FUNCTION_BLOCK FB_Machine EXTENDS FB_Generic
VAR_INPUT
	pPML_Instance1	: POINTER TO FB_Generic;
	pPML_Instance2	: POINTER TO FB_Generic;//instance for couple and uncouple
	pPackTags		: POINTER TO ST_PackMLv30;
	pSafetySystem	: POINTER TO FB_Safety_Subsystem;
END_VAR
VAR_OUTPUT

END_VAR
VAR	
	stSubModuleInfo		: ARRAY [1..iSubModule] OF ST_PMLSubUnitInfo;	//Informations about the Subunits
//	pPML_Instance	: ARRAY [1..iSubModule] OF POINTER TO FB_Generic;
	arrCouple	: ARRAY [1..iSubModule] OF BOOL;
	arrCmd		: ARRAY [1..iSubModule] OF E_PMLCommand;
	unCouple	: BOOL;//all modules uncoupling
	
	rtrig_alarm	:ARRAY [1..iSubModule] OF ARRAY[1..MaxAlarms] OF R_TRIG;
	
	iCmd_unitsActive	: INT;
	iCmd_transfer	: INT;


	preEstate	: E_PMLState;
	
END_VAR
VAR CONSTANT
	iSubModule	: UINT :=2;
END_VAR

//pPML_Instance[1]	:= ADR(GVL.fb_sample1);
//pPML_Instance[2]	:= ADR(GVL.fb_sample2);
///////////////////////////////////////////for signal system/////////////////////////////////////////////////////////////
IF NOT unCouple THEN
	FOR i:=1 TO UINT_TO_INT(iSubModule) DO
		arrCmd[i]:=eCommand;
		arrCouple[i]:= TRUE;
//		pPML_Instance[i]^._bCouple	:= TRUE;

	END_FOR
END_IF
unCouple	:= TRUE;//for mix sysytem
//////////////////////////////////////////////couple cmd//////////////////////////////////////////////////////////
//FOR i:=1 TO UINT_TO_INT(iSubModule) DO
//	IF arrCouple[i] THEN
//		arrCmd[i]:=eCommand;
//	END_IF
//END_FOR

CASE iCmd_transfer OF	
	0:
		IF eCommand<>ePMLCommand_Undefined THEN
			iCmd_transfer	:= 1;
		END_IF
	1:	
		IF arrCouple[1] THEN
			arrCmd[1]	:= eCommand;
		END_IF
		IF arrCouple[2] THEN
			arrCmd[2]	:= eCommand;
		END_IF
		iCmd_transfer	:= 2;	
	2:
		CASE preEstate OF
			ePMLState_Undefined:
				IF eState=ePMLState_Aborted THEN
					iCmd_transfer	:= 3;
				END_IF			
			ePMLState_Aborted,ePMLState_Clearing:
				IF eState=ePMLState_Stopped OR eState=ePMLState_Aborted THEN
					iCmd_transfer	:= 3;
				END_IF
			ePMLState_Stopped,ePMLState_Resetting:
				IF eState=ePMLState_Idle OR eState=ePMLState_Aborted THEN
					iCmd_transfer	:= 3;
				END_IF				
			ePMLState_Idle,ePMLState_Starting:
				IF eState=ePMLState_Execute OR eState=ePMLState_Stopped OR eState=ePMLState_Aborted THEN
					iCmd_transfer	:= 3;
				END_IF				
			ePMLState_Execute,ePMLState_Aborting,ePMLState_Stopping:
				IF eState=ePMLState_Stopped OR eState=ePMLState_Aborted THEN
					iCmd_transfer	:= 3;
				END_IF				
		END_CASE	
	3:
		arrCouple[2]	:= FALSE;
		arrCmd[1]	:=	ePMLCommand_Undefined;
		arrCmd[2]	:=	ePMLCommand_Undefined;
		iCmd_transfer	:= 0;	
END_CASE



pPML_Instance1^(
	eModeCommand:= eModeCommand, 
	eCommand:= arrCmd[1], 
	eMode=> , 
	eState=> stSubModuleInfo[1].eState, 
	bUndefinedDone=> , 
	bInvalidModeCommandOut=> , 
	bChangeIntoProduction=> );
stSubModuleInfo[1].Active		:= arrCouple[1];

pPML_Instance2^(
	eModeCommand:= eModeCommand, 
	eCommand:= , 
	eMode=> , 
	eState=> stSubModuleInfo[2].eState, 
	bUndefinedDone=> , 
	bInvalidModeCommandOut=> , 
	bChangeIntoProduction=> );
IF stSubModuleInfo[2].Active THEN
	pPML_Instance2^.eCommand	:= arrCmd[2];
END_IF	
stSubModuleInfo[2].Active		:= arrCouple[2];


IF  pPML_Instance1^.bUndefinedDone AND 
	pPML_Instance2^.bUndefinedDone 
THEN
	bUndefinedDone := TRUE;
END_IF

//The fbStateMachine from FB_Machine gets the Information about the states and activity from the subunits
fbStateMachine.stSubUnitInfoRef.ArraySize		:= SIZEOF(stSubModuleInfo);
fbStateMachine.stSubUnitInfoRef.NoOfSubUnits	:= iSubModule;
fbStateMachine.stSubUnitInfoRef.pArray			:= ADR(stSubModuleInfo);



//Set unit information 
M_SetUnitInfo();






SUPER^();

{attribute 'object_name' := 'M_Clearing'}
METHOD M_Clearing

CASE fbUnitModeManager.eModeStatus OF
	ePMLProtUnitMode_Production:		//Production, Mantainance, Manual
		FOR i:=1 TO 3 DO//try clear alarm several times
			FOR j:=1 TO MaxAlarms DO
				GVL.pml_adminAlarm.M_AcknowledgeAlarm(stAdmin:=pPackTags^.Admin,stAlarm:=pPackTags^.Admin.Alarm[j]);
				GVL.pml_adminAlarm.M_ClearAlarm(stAdmin:=pPackTags^.Admin,stAlarm:=pPackTags^.Admin.Alarm[j]);
			END_FOR	
		END_FOR	
		IF pSafetySystem^.M_reset() THEN
			IF pSafetySystem^.xError THEN
				IF M_UnitsActive(ePMLCommand_Abort)THEN
					eCommand	:= ePMLCommand_Abort;
				END_IF
			ELSE
				M_StateComplete();
			END_IF
		END_IF	
		
	
	ePMLProtUnitMode_Maintenance, ePMLProtUnitMode_Manual, ePMLUnitMode_Service:
		M_StateComplete();
END_CASE
END_METHOD

{attribute 'object_name' := 'M_Execute'}
METHOD M_Execute
END_METHOD

{attribute 'object_name' := 'M_Resetting'}
METHOD M_Resetting
CASE fbUnitModeManager.eModeStatus OF
	ePMLProtUnitMode_Production:		//Production, Mantainance, Manual	
		IF pSafetySystem^.M_reset() THEN
			IF pSafetySystem^.xError THEN
				IF M_UnitsActive(ePMLCommand_Abort)THEN
					eCommand	:= ePMLCommand_Abort;
				END_IF
			ELSE
				M_StateComplete();
			END_IF
		END_IF	
		
	
	ePMLProtUnitMode_Maintenance, ePMLProtUnitMode_Manual, ePMLUnitMode_Service:
		M_StateComplete();
END_CASE
END_METHOD

METHOD M_SetUnitInfo
VAR_INPUT
END_VAR
GVL.aUnitInfo[eMachine].Name			:= 'fbMachine';
GVL.aUnitInfo[eMachine].ActMode			:= eMode;
GVL.aUnitInfo[eMachine].ActState		:= eState;

GVL.aUnitInfo[eWorking1].Name			:= GVL.fb_working1._sInstanceName;
GVL.aUnitInfo[eWorking1].ActMode		:= GVL.fb_working1.eMode;
GVL.aUnitInfo[eWorking1].ActState		:= GVL.fb_working1.eState;

GVL.aUnitInfo[eLoading].Name			:= GVL.fb_loading._sInstanceName;
GVL.aUnitInfo[eLoading].ActMode			:= GVL.fb_loading.eMode;
GVL.aUnitInfo[eLoading].ActState		:= GVL.fb_loading.eState;

GVL.aUnitInfo[eWorking2].Name			:= GVL.fb_working2._sInstanceName;
GVL.aUnitInfo[eWorking2].ActMode		:= GVL.fb_working2.eMode;
GVL.aUnitInfo[eWorking2].ActState		:= GVL.fb_working2.eState;
END_METHOD

{attribute 'object_name' := 'M_Starting'}
METHOD M_Starting
CASE fbUnitModeManager.eModeStatus OF
	ePMLProtUnitMode_Production:		//Production, Mantainance, Manual
		//Resetting all Commands and Value
		G_HMI.bAging_test	:= FALSE;
		M_StateComplete();
	ePMLProtUnitMode_Maintenance, ePMLProtUnitMode_Manual, ePMLUnitMode_Service:
		M_StateComplete();
END_CASE
END_METHOD

//nomal
//idle/excute->stop 	idle/excute->abort
//loding error->abort
METHOD M_UnitsActive : BOOL
VAR_INPUT
	preCmd	: E_PMLCommand;
END_VAR
VAR 
	
END_VAR
M_UnitsActive	:= FALSE;




CASE iCmd_unitsActive OF
	0:
		iCmd_unitsActive	:= 1;
		iCmd_transfer	:= 0;
//get the command from main
	1:
		iCmd_unitsActive	:= 2;
//verify state
	2:
		IF NOT pSafetySystem^.xEstop THEN//no matter in which state,couple all the units
			arrCouple[1]	:= TRUE;
			arrCouple[2]	:= TRUE;	
			iCmd_unitsActive	:= 4;		
		ELSE
			IF (stSubModuleInfo[1].eState=ePMLState_Aborted OR stSubModuleInfo[1].eState=ePMLState_Stopped OR
				stSubModuleInfo[1].eState=ePMLState_Idle OR stSubModuleInfo[1].eState=ePMLState_Execute) AND
				(stSubModuleInfo[2].eState=ePMLState_Aborted OR stSubModuleInfo[2].eState=ePMLState_Stopped OR
				stSubModuleInfo[2].eState=ePMLState_Idle OR stSubModuleInfo[2].eState=ePMLState_Execute) AND
				(eState=ePMLState_Aborted OR eState=ePMLState_Stopped OR eState=ePMLState_Idle OR eState=ePMLState_Execute)
			THEN
				iCmd_unitsActive	:= 3;
			END_IF
		END_IF
//determine if couple or not
	3:
		CASE stSubModuleInfo[1].eState OF
			ePMLState_Aborted:
				CASE stSubModuleInfo[2].eState OF
					ePMLState_Aborted:
						CASE preCmd OF
							ePMLCommand_Clear:
								arrCouple[1]	:= TRUE;
								arrCouple[2]	:= TRUE;	
							ePMLCommand_Reset:	
								//					
							ePMLCommand_Start:	
								//
							ePMLCommand_Stop:	
								//
							ePMLCommand_Abort:
								IF pPML_Instance2^.isError OR pSafetySystem^.xEstop_behavior THEN
									arrCouple[2]	:= TRUE;
								ELSE
									arrCouple[2]	:= FALSE;
								END_IF									
						END_CASE						
					ePMLState_Stopped:
						CASE preCmd OF
							ePMLCommand_Clear:
								arrCouple[1]	:= TRUE;
								arrCouple[2]	:= FALSE;	
							ePMLCommand_Reset:	
								//					
							ePMLCommand_Start:	
								//
							ePMLCommand_Stop:	
								//
							ePMLCommand_Abort:
								IF pPML_Instance2^.isError OR pSafetySystem^.xEstop_behavior THEN
									arrCouple[2]	:= TRUE;
								ELSE
									arrCouple[2]	:= FALSE;
								END_IF									
						END_CASE					
					ePMLState_Idle:
						CASE preCmd OF
							ePMLCommand_Clear:
								arrCouple[1]	:= TRUE;
								arrCouple[2]	:= FALSE;	
							ePMLCommand_Reset:	
								//					
							ePMLCommand_Start:	
								//
							ePMLCommand_Stop:	
								//
							ePMLCommand_Abort:
								IF pPML_Instance2^.isError OR pSafetySystem^.xEstop_behavior THEN
									arrCouple[2]	:= TRUE;
								ELSE
									arrCouple[2]	:= FALSE;
								END_IF									
						END_CASE
					ePMLState_Execute:
						CASE preCmd OF
							ePMLCommand_Clear:
								arrCouple[1]	:= TRUE;
								arrCouple[2]	:= FALSE;	
							ePMLCommand_Reset:	
								//					
							ePMLCommand_Start:	
								//
							ePMLCommand_Stop:	
								//
							ePMLCommand_Abort:
								IF pPML_Instance2^.isError OR pSafetySystem^.xEstop_behavior THEN
									arrCouple[2]	:= TRUE;
								ELSE
									arrCouple[2]	:= FALSE;
								END_IF									
						END_CASE	
				END_CASE		
			ePMLState_Stopped:
				CASE stSubModuleInfo[2].eState OF	
					ePMLState_Aborted:
						//
					ePMLState_Stopped:
						CASE preCmd OF
							ePMLCommand_Clear:
								//
							ePMLCommand_Reset:	
								arrCouple[1]	:= TRUE;
								arrCouple[2]	:= TRUE;						
							ePMLCommand_Start:	
								//
							ePMLCommand_Stop:	
								//
							ePMLCommand_Abort:
								IF pPML_Instance2^.isError OR pSafetySystem^.xEstop_behavior THEN
									arrCouple[2]	:= TRUE;
								ELSE
									arrCouple[2]	:= FALSE;
								END_IF									
						END_CASE					
					ePMLState_Idle:
						CASE preCmd OF
							ePMLCommand_Clear:
								//
							ePMLCommand_Reset:	
								arrCouple[1]	:= TRUE;
								arrCouple[2]	:= FALSE;						
							ePMLCommand_Start:	
								//
							ePMLCommand_Stop:	
								//
							ePMLCommand_Abort:
								IF pPML_Instance2^.isError OR pSafetySystem^.xEstop_behavior THEN
									arrCouple[2]	:= TRUE;
								ELSE
									arrCouple[2]	:= FALSE;
								END_IF									
						END_CASE					
					ePMLState_Execute:
						CASE preCmd OF
							ePMLCommand_Clear:
								//
							ePMLCommand_Reset:	
								arrCouple[1]	:= TRUE;
								arrCouple[2]	:= FALSE;						
							ePMLCommand_Start:	
								//
							ePMLCommand_Stop:	
								//
							ePMLCommand_Abort:
								IF pPML_Instance2^.isError OR pSafetySystem^.xEstop_behavior THEN
									arrCouple[2]	:= TRUE;
								ELSE
									arrCouple[2]	:= FALSE;
								END_IF									
						END_CASE					
				END_CASE	

	
			ePMLState_Idle:
				CASE stSubModuleInfo[2].eState OF	
					ePMLState_Aborted:
						//
					ePMLState_Stopped:
						//
					ePMLState_Idle:
						CASE preCmd OF
							ePMLCommand_Clear:
								//
							ePMLCommand_Reset:	
								//						
							ePMLCommand_Start:	
								arrCouple[1]	:= TRUE;
								arrCouple[2]	:= TRUE;
							ePMLCommand_Stop:	
								arrCouple[1]	:= TRUE;
								arrCouple[2]	:= FALSE;									
							ePMLCommand_Abort:
								IF pPML_Instance2^.isError OR pSafetySystem^.xEstop_behavior THEN
									arrCouple[2]	:= TRUE;
								ELSE
									arrCouple[2]	:= FALSE;
								END_IF									
						END_CASE					
					ePMLState_Execute:
						CASE preCmd OF
							ePMLCommand_Clear:
								//
							ePMLCommand_Reset:	
								//						
							ePMLCommand_Start:	
								arrCouple[1]	:= TRUE;
								arrCouple[2]	:= FALSE;
							ePMLCommand_Stop:	
								arrCouple[1]	:= TRUE;
								arrCouple[2]	:= FALSE;									
							ePMLCommand_Abort:
								IF pPML_Instance2^.isError OR pSafetySystem^.xEstop_behavior THEN
									arrCouple[2]	:= TRUE;
								ELSE
									arrCouple[2]	:= FALSE;
								END_IF									
						END_CASE
				END_CASE	
			ePMLState_Execute:
				CASE stSubModuleInfo[2].eState OF	
					ePMLState_Aborted:
						//
					ePMLState_Stopped:
						//
					ePMLState_Idle:
						//
					ePMLState_Execute:
						CASE preCmd OF
							ePMLCommand_Clear:
								//
							ePMLCommand_Reset:	
								//						
							ePMLCommand_Start:	
								//
							ePMLCommand_Stop:	
								arrCouple[1]	:= TRUE;
								arrCouple[2]	:= FALSE;									
							ePMLCommand_Abort:
								IF pPML_Instance2^.isError OR pSafetySystem^.xEstop_behavior THEN
									arrCouple[2]	:= TRUE;
								ELSE
									arrCouple[2]	:= FALSE;
								END_IF									
						END_CASE	
				END_CASE	
		END_CASE
		iCmd_unitsActive	:= 4;
		
	4:
		preEstate	:= eState;
		iCmd_unitsActive	:= 0;
		M_UnitsActive	:= TRUE	;
	
//set the command to units
END_CASE
END_METHOD

END_FUNCTION_BLOCK

(* stored: Version 1.1.0.1, ProductVersion 3.1.4024.12
   POU FB_Machine: Id {8f8b4044-4b54-4b05-9dcb-51655cce136f}, SpecialFunc None
   Method M_Clearing: Id {242a7bec-354c-403a-8360-5cddeab3cb27}
   Method M_Execute: Id {41e5f6e5-a4a2-4dc8-bbd5-97eabfb821d3}
   Method M_Resetting: Id {c82aab94-be7d-4f8e-a811-07458a877516}
   Method M_SetUnitInfo: Id {1ffbecee-8eda-4bb4-8a81-6dafcd0ad308}
   Method M_Starting: Id {607735ee-5540-4bee-8bb9-efaec3726053}
   Method M_UnitsActive: Id {7bdd32b7-6eb3-45fa-829d-2018203ee44d} *)
